PROGRAM PRG_LVCP5_PowerMeasurement
VAR
	// Enerji Yönetimi
	fbEL3453	: FB_EL3453;	
	stEL3453	: stEL3453;
END_VAR


	fbEL3453(pOut := ADR(stEL3453));

END_PROGRAM

(* stored: Version 1.1.0.1, ProductVersion 3.1.4024.15
   POU PRG_LVCP5_PowerMeasurement: Id {9d98de9f-f3fc-4a9c-8413-8f8cfb40b303}, SpecialFunc None *)
